// TIA Portal project "ProyectoAutomatizacion2_MarioBetancourt" (V20)

(* hardware
DEVICE "S7-300/ET200M station_1"  S7-300 station
   slot 0: "Rail_0"  Rail  6ES7 390-1***0-0AA0
   slot 2: "PLC_1"  CPU 315-2 DP  6ES7 315-2AH14-0AB0  V3.0
      slot 0: "MPI interface_1"  MPI
      slot 1: "DP interface_1"  DP
   slot 4: "AI 8x12BIT_1"  AI8 x 12 bits  6ES7 331-7KF02-0AB0
   slot 5: "AO 8x12BIT_1"  AO8 x 12 bits  6ES7 332-5HF00-0AB0
   slot 6: "DI 16x24VDC_1"  DI16 x 24VDC  6ES7 321-1BH02-0AA0
   slot 7: "DO 16x24VDC/0.5A_1"  DO16 x 24VDC / 0.5A  6ES7 322-1BH01-0AA0
*)

// ===== PLC "PLC_1"  CPU 315-2 DP =====

VAR_GLOBAL   // PLC tag table "Default tag table"
   "BotonVerde" AT %I8.0 : Bool;   // Marcha general de la línea
   "BotonRojo" AT %I8.1 : Bool;   // Paro general de la línea
   "SelectorIzquierda" AT %I8.2 : Bool;   // Sin uso funcional en este proyecto
   "SelectorDerecha" AT %I8.3 : Bool;   // Sin uso funcional en este proyecto
   "ParoEmergencia" AT %I8.4 : Bool;   // E-stop: abortar de inmediato y forzar estado seguro
   "SensorOptico" AT %I9.0 : Bool;   // Dispara el conteo de 3 y la carga de la posición 0 del shift register
   "SensorPaso" AT %I9.1 : Bool;   // Genera el pulso de avance que desplaza el shift register
   "SensorVerificacion1" AT %I9.2 : Bool;   // Mide el nivel de llenado de la botella en la estación E-1
   "SensorVerificacion2" AT %I9.3 : Bool;   // Mide el nivel de llenado de la botella en la estación E-2
   "SensorVerificacion3" AT %I9.4 : Bool;   // Mide el nivel de llenado de la botella en la estación E-3
   "SensorRTD" AT %IW272 : Int;   // Interbloqueo obligatorio de temperatura
   "MotorBanda" AT %Q12.0 : Bool;   // Avance de la banda / desplazamiento del shift register
   "ActuadorLlenado1" AT %Q12.1 : Bool;   // Válvula/dosificador, habilitado solo con temperatura en rango
   "ActuadorLlenado2" AT %Q12.2 : Bool;   // Válvula/dosificador, habilitado solo con temperatura en rango
   "ActuadorLlenado3" AT %Q12.3 : Bool;   // Válvula/dosificador, habilitado solo con temperatura en rango
   "ActuadorRechazo" AT %Q12.4 : Bool;   // Expulsión de producto defectuoso fuera de la banda
   "BalizaMarcha" AT %Q12.5 : Bool;   // Encendida mientras el sistema opera en automático
   "BalizaAlarmaTemperatura" AT %Q12.6 : Bool;   // Encendida mientras el llenado está bloqueado por el RTD
   "BalizaLoteCompleto" AT %Q12.7 : Bool;   // Encendida al alcanzar el lote objetivo de producto bueno
   "MarcaSeguridad" AT %M20.0 : Bool;   // Marca global de seguridad. Activada desde FC1.
   "MarcaTemperatura" AT %M20.1 : Bool;   // Marca de habilitación de llenado por interbloqueo por temperatura (HabilitaLlenado)
END_VAR

DATA_BLOCK "DB_ShiftRegister"   // DB50
TITLE = Registro de desplazamiento
{ S7_Optimized_Access := 'FALSE' }
VERSION : 0.1
// Data Block para monitorear el estado de los productos en tránsito sobre la banda.
   VAR
      ShiftRegister : Array[0..19] of Int;
   END_VAR
BEGIN
END_DATA_BLOCK

DATA_BLOCK "DB_Config"   // DB100
TITLE = Bloque de datos de configuración
{ S7_Optimized_Access := 'FALSE' }
VERSION : 0.1
// Contiene parámetros generales para el sistema de automatización.
   VAR
      TempMin : Real;   // Límite inferior de temperatura válida para llenado
      TempMax : Real;   // Límite superior de temperatura válida para llenado
      TiempoLlenado : Time;   // Duración del pulso de llenado en cada estación
      UmbralNivelOK : Real;   // Umbral de distancia de nivel que define "llenado correcto"
      LoteObjetivo : Int;   // Cantidad de producto buenoq ue define un lote completo
   END_VAR
BEGIN
END_DATA_BLOCK

DATA_BLOCK "DB_IoT"   // DB200
TITLE = DB IoT
{ S7_Optimized_Access := 'FALSE' }
VERSION : 0.1
// Interfaz de intercambio con MATLAB, no optimizado
BEGIN
END_DATA_BLOCK

FUNCTION_BLOCK "FB_Secuenciador"   // FB1, STL
TITLE = FB Secuenciador
{ S7_Optimized_Access := 'FALSE' }
VERSION : 0.1
// Máquina de estados de la Sección 5.5(Espera, Conteo, Paro, EsperaTemperatura, Llenando, Reanudando). Instancia única.
   VAR_INPUT
      boton_verde : Bool;
      paro_emergencia : Bool;
      sensor_optico : Bool;
      sensor_paso : Bool;
      contador_detecciones : Counter;
      interbloqueo_temperatura_activo : Bool;
      nivel_llenado_ok : Bool;
      tiempo_llenado_E1 : S5Time;
      tiempo_llenado_E2 : S5Time;
      tiempo_llenado_E3 : S5Time;
   END_VAR
   VAR_OUTPUT
      motor_banda : Bool;
      baliza_temperatura : Bool;
      actuador_llenado1 : Bool;
      actuador_llenado2 : Bool;
      actuador_llenado3 : Bool;
   END_VAR
   VAR
      paso0_espera : Bool;   // Marca de paso 0 - Estado Inicial / Reposo
      paso1_conteo : Bool;   // Marca de paso 1 - avanzando banda y contando botellas
      paso2_paro_temp_check : Bool;   // Marca de paso 2 - Banda detenida, verificando RTD
      paso3_llenado : Bool;   // Marca de paso 3 - Llenado activo
      paso4_reanudando : Bool;   // Marca de paso 4 - Llenado completo, reanudando banda
      contador_botellas : Int;   // Conteo de botellas ingresadas
      memoria_flanco_optico : Bool;   // Memoria de flanco
   END_VAR
BEGIN

REGION Network 1: Inicialización del Secuenciador
   // Si al energizar la CPU ningún paso está activo, activar la marca del paso 0 (reposo)
         AN    #paso0_espera;
         AN    #paso1_conteo;
         AN    #paso2_paro_temp_check;
         AN    #paso3_llenado;
         AN    #paso4_reanudando;
         S     #paso0_espera;
END_REGION

REGION Network 2: Paso 0 - Reposo (Transición de Entrada)
   // Fin de Ciclo o Reset -> Paso 0
         A     #paso4_reanudando;
         S     #paso0_espera;
         R     #paso4_reanudando;
END_REGION

REGION Network 3: Paso 0 - Reposo (Network de Acción)
   // Mientras el sistema está en reposo, el contador de botellas se mantiene ne cero.
         A     #paso0_espera;
         R     #contador_detecciones;
END_REGION

REGION Network 4: Paso 0 - Reposo (Transición de Salida)
   // Si el botón verde (%I8.0) está presionado y el paro de emergencia (NC) está cerrado, transicionar hacia el paso 1 (Inicio de Marcha)
         A     #paso0_espera;
         A     #boton_verde;
         A     #paro_emergencia;
         S     #paso1_conteo;
         R     #paso0_espera;
END_REGION

REGION Network 5: Paso 1 - Conteo de 3 botellas (Network de Acción)
   // Energizar la banda (%Q12.0) e incrementar el contador con cada flanco del sensor óptico.
   // Encender el motor si la marca del paso 1 es 1
         A     #paso1_conteo;
         S     #motor_banda;

   // Detección de flanco positivo del sensor óptico
   // e incremento del contador de detecciones
         A     #paso1_conteo;
         A     #sensor_optico;
         CU    #contador_detecciones;
END_REGION

REGION Network 6: Paso 1 - Conteo de botellas (Transición de Salida)
   // Si se detectan tres botellas, transicionar a  Paso 2 (Chequeo de Temperatura de RTD).
         A     #paso1_conteo;
         JCN   M003;

   // Transicionar sólo cuando ya se hayan contador 3 botellas
         L     #contador_detecciones;
         L     3;
         >=I;
         S     #paso2_paro_temp_check;
         R     #paso1_conteo;

   M003: NOP   0;
END_REGION

REGION Network 7: Paso 2 - Paro de Banda e Interbloqueo de Temperatura (Network de Acción)
   // Detener la banda siempre que este estado se encuentre activo.
   // Detener la banda y encender baliza si el interbloqueo de temperatura
   // está activo (señal controlada por FC2)
         A     #paso2_paro_temp_check;
         R     #motor_banda;
         A     #interbloqueo_temperatura_activo;
         A     #baliza_temperatura;
END_REGION

REGION Network 8: Paso 2 - Paro de Banda e Interbloqueo de Temperatura (Transición de Salida).
   // Transicionar del paso 2 al paso 3 si el bit de habilitación de temperatura "DB_Config.HabilitaLlenado" es 1
   // Transicionar cuando el interbloqueo se haya desactivado
         A     #paso2_paro_temp_check;
         AN    #interbloqueo_temperatura_activo;
         S     #paso3_llenado;
         R     #paso2_paro_temp_check;
END_REGION

REGION Network 9: Paso 3 - Llenado activo simultáneo (Network de Acción)
   // Mientras este paso está activo, activar los actuadores de las tres estaciones de llenado.
         A     #paso3_llenado;
         =     #actuador_llenado1;
         =     #actuador_llenado2;
         =     #actuador_llenado3;
END_REGION

REGION Network 10: Paso 3 - Llenado activo simultaneo (Transición de Salida)
   // Si las 3 estaciones completan su tiempo de llenado, transicionar hacia el paso 4
         A     #paso3_llenado;
         A     #nivel_llenado_ok;  // Señal de FC4
         S     #paso4_reanudando;
         R     #paso3_llenado;
END_REGION

REGION Network 11: Paso 4 - Reanudación de banda (Network de acción)
   // Reestablecer señales de llenado y reanudar marcha. La network de transición es la network 2.
   // Continuar sólo si el paso está activo
         A     #paso4_reanudando;
         S     #motor_banda;

   // Si la marca de paso está activa, reiniciar el contador a 0
         A     #paso4_reanudando;
         R     #contador_detecciones;
END_REGION
END_FUNCTION_BLOCK

FUNCTION_BLOCK "FB_Estacion_Llenado"   // FB2, LAD
TITLE = FB Estación Llenado
{ S7_Optimized_Access := 'FALSE' }
VERSION : 0.1
// Lógica genérica de una estación de llenado: temporiza-
// dor, gate de HabilitaLlenado, actualización de estado
// en DB50. Sin referencias a una instancia específica.
BEGIN
END_FUNCTION_BLOCK

FUNCTION "FC_Seguridad" : Void   // FC1, STL
TITLE = FC Seguridad
{ S7_Optimized_Access := 'FALSE' }
VERSION : 0.1
// Paro de emergencia. Fuerza todas las salidas de potencia a 0 y lleva al secuenciador a estado seguro. Se ejecuta siempre primero.
   VAR_INPUT
      paro_emergencia : Bool;
   END_VAR
   VAR_OUTPUT
      motor_banda : Bool;
      actuador_llenado_e1 : Bool;
      actuador_llenado_e2 : Bool;
      actuador_llenado_e3 : Bool;
      actuador_rechazo : Bool;
   END_VAR
   VAR_TEMP
      marca_flanco_positivo : Bool;
      marca_flanco_negativo : Bool;
   END_VAR
BEGIN

REGION Network 1: Paro de Emergencia
   // Si el paro de emergencia (NC) se abre, forzar todas las salidas a 0. Si el paro está cerrado, NO HACER NADA.
   // Leer paro (1 = seguro, 0 = presionado)
         A     #paro_emergencia;
         JC    NO_HACER_NADA;

   // --- ZONA DE EMERGENCIA ---
   // Este bloque se ejecuta sólo si el botón
   // fue presionado
         CLR;  // Pone el RLO forzadamente en 0
         =     #motor_banda;
         =     #actuador_llenado_e1;
         =     #actuador_llenado_e2;
         =     #actuador_llenado_e3;
         =     #actuador_rechazo;

   NO_HACER_NADA:NOP   0;
END_REGION
END_FUNCTION

FUNCTION "FC_Interbloqueo_Temp" : Void   // FC2, STL
TITLE = FC Interbloqueo por Exceso de Temperatura
{ S7_Optimized_Access := 'FALSE' }
VERSION : 0.1
// Esta función lee %PIW272, compara contra DB_Config, escribe HabilitaLlenado y %Q12.6
   VAR_INPUT
      raw_temp : Int;
      temp_min : Real;
      temp_max : Real;
   END_VAR
   VAR_OUTPUT
      temp_actual : Real;
      interbloqueo_temp_activo : Bool;
   END_VAR
   VAR_TEMP
      temp_real : Real;
   END_VAR
   VAR CONSTANT
      factor_escala : Real := 10.0;
   END_VAR
BEGIN

REGION Network 1: Conversión de lectura analógica (INT) a REAL (°C)
         L     #raw_temp;  // Carga temperatura
         ITD;  // Conversión INT a DOUBLE
         DTR;  // Conversión DOUBLE a REAL
         L     #factor_escala;  // Cargar factor de escala (cte)
         /R;  // División real
         T     #temp_real;  // Guardar en variable local
         T     #temp_actual;  // Guardar en variable de salida
END_REGION

REGION Network 2: Verificación de rango e interbloqueo seguro
   // Evaluar si la Temperatura >= Temperatura Mínima
         L     #temp_real;
         L     #temp_min;
         >=R;
         JCN   TEMP_INTERLOCK;  //Si es menor, bloquear

   // Evaluar si Temperatura <= Temperatura Máxima
         L     #temp_real;
         L     #temp_max;
         <=R;
         JCN   TEMP_INTERLOCK;

   // Si la temperatura está dentro del rango seguro
         CLR;  // Hace que RLO = 0
         =     #interbloqueo_temp_activo;
         JU    FC2_END;  // Salta hacia el final

   // Si la temperatura está fuera del rango seguro
   TEMP_INTERLOCK:NOP   0;
         SET;
         =     #interbloqueo_temp_activo;  // Encender interbloqueo

   FC2_END:NOP   0;
END_REGION
END_FUNCTION

FUNCTION "FC_Shift_Register" : Void   // FC3, FBD
TITLE = FC Shift Register
{ S7_Optimized_Access := 'FALSE' }
VERSION : 0.1
// Implementa el desplazamiento de DB50 en cada pulso 
// de %I9.1
   VAR_INPUT
      pulse_encoder : Bool;   // Señal de avance
      sensor_optico : Bool;   // Sensor de presencia a la entrada
   END_VAR
   VAR_IN_OUT
      flanco_memoria : Bool;   // Bit para detección de flanco positivo
      posicion : Array[0..1] of Int;   // Arreglo del shift register
   END_VAR
   VAR_TEMP
      db_num : Word;
      index : Int;
      pos_edge : Bool;
      offset : DWord;
   END_VAR
BEGIN
END_FUNCTION

FUNCTION "FC_Verificacion" : Void   // FC4, STL
TITLE = FC Verificación
{ S7_Optimized_Access := 'FALSE' }
VERSION : 0.1
// Lee %I10.0– %I10.2, compara contra UmbralNivelOK,
// actualiza estados 3/4 en las posiciones 10–12 de D
BEGIN
END_FUNCTION

FUNCTION "FC_Rechazo_Conteo" : Void   // FC5, STL
TITLE = FC Rechazo Conteo
{ S7_Optimized_Access := 'FALSE' }
VERSION : 0.1
// Lee posición 17 de DB50, acciona %Q12.4
// si aplica; en posición 18, actualiza
// DB_IoT.ConteoBuenos/ConteoRechazados.
BEGIN
END_FUNCTION

FUNCTION "FC_Enlace_Snap7" : Void   // FC6, STL
TITLE = FC Enlace Snap7
{ S7_Optimized_Access := 'FALSE' }
VERSION : 0.1
BEGIN
END_FUNCTION

ORGANIZATION_BLOCK "Main"   // OB1, STL
TITLE = "Main Program Sweep (Cycle)"
{ S7_Optimized_Access := 'FALSE' }
VERSION : 0.1
   VAR_TEMP
      OB1_EV_CLASS : Byte;   // Bits 0-3 = 1 (Coming event), Bits 4-7 = 1 (Event class 1)
      OB1_SCAN_1 : Byte;   // 1 (Cold restart scan 1 of OB 1), 3 (Scan 2-n of OB 1)
      OB1_PRIORITY : Byte;   // Priority of OB Execution
      OB1_OB_NUMBR : Byte;   // 1 (Organization block 1, OB1)
      OB1_RESERVED_1 : Byte;   // Reserved for system
      OB1_RESERVED_2 : Byte;   // Reserved for system
      OB1_PREV_CYCLE : Int;   // Cycle time of previous OB1 scan (milliseconds)
      OB1_MIN_CYCLE : Int;   // Minimum cycle time of OB1 (milliseconds)
      OB1_MAX_CYCLE : Int;   // Maximum cycle time of OB1 (milliseconds)
      OB1_DATE_TIME : Date_And_Time;   // Date and time OB1 started
   END_VAR
BEGIN

REGION Network 1: FC Seguridad
         CALL  "FC_Seguridad"
         ( paro_emergencia     := "ParoEmergencia",
           motor_banda         := "MotorBanda",
           actuador_llenado_e1 := "ActuadorLlenado1",
           actuador_llenado_e2 := "ActuadorLlenado2",
           actuador_llenado_e3 := "ActuadorLlenado3",
           actuador_rechazo    := "ActuadorRechazo"
         );
END_REGION
END_ORGANIZATION_BLOCK